INTERFACE PUBLIC I_MoveAbsoluteBuilder EXTENDS __System.IQueryInterface

METHOD PUBLIC Acceleration : I_MoveBuilder
VAR_INPUT
	value : LREAL;
END_VAR
END_METHOD

METHOD PUBLIC BufferMode : I_MoveBuilder
VAR_INPUT
	mode : AxisBufferMode;
END_VAR
END_METHOD

METHOD PUBLIC BuildMoveAbsoluteCommand : I_MoveCommand
END_METHOD

METHOD PUBLIC Deceleration : I_MoveBuilder
VAR_INPUT
	value : LREAL;
END_VAR
END_METHOD

METHOD PUBLIC Jerk : I_MoveBuilder
VAR_INPUT
	value : LREAL;
END_VAR
END_METHOD

METHOD PUBLIC Position : I_MoveAbsoluteBuilder
VAR_INPUT
	value : LREAL;
END_VAR
END_METHOD

METHOD PUBLIC Velocity : I_MoveBuilder
VAR_INPUT
	value : LREAL;
END_VAR
END_METHOD

END_INTERFACE

(* stored: Version 1.1.0.1, ProductVersion 3.1.4024.12
   Itf I_MoveAbsoluteBuilder: Id {5079e367-9935-04a9-3dba-01451a92a74a}
   Method Acceleration: Id {156df490-e1dc-0676-318f-a2186da883d8}
   Method BufferMode: Id {c52a5773-32c4-0146-24bd-043678112a2e}
   Method BuildMoveAbsoluteCommand: Id {4c34f79d-c64b-0824-3130-35aa512d84ab}
   Method Deceleration: Id {e81250ab-a25a-07ce-3b79-64dfb2686766}
   Method Jerk: Id {04965531-bfb8-0df7-06ef-e84ed27dce8d}
   Method Position: Id {8139d982-0eac-007c-3859-939e66315c65}
   Method Velocity: Id {2dd2d8f6-cf68-0cb7-0f3d-a9c5726588eb} *)
